TYPE ST_PowerMonitor_get :
STRUCT
	PQMeterReady	: 	BOOL;
	InputField		:	ST_PowerMonitor_InputField;	
	OutputField		:	ST_PowerMonitor_OutputField;
	InternalSupply	:	ST_PowerMonitor_Internal;
	
	//Inverter power/energy input & output
	BESS			:	ST_PowerMonitor_BESS;

	
	events			:	ST_PowerMonitor_Events;
END_STRUCT
END_TYPE

(* stored: Version 1.1.0.1, ProductVersion 3.1.4024.12
   DUT ST_PowerMonitor_get: Id {23aaa03f-abd8-4194-9474-ce74b9a36cd6} *)
